FUNCTION_BLOCK FB_AnalogueInputBase IMPLEMENTS IAnalogueInput
VAR_INPUT
END_VAR
VAR_OUTPUT
END_VAR
VAR
	_processData : REFERENCE TO AnalogueStatus;
	_signalType : DINT;
	_resolution : DINT;
END_VAR

PROPERTY PUBLIC Error : bool
GET
Error := _processData.Underrange OR _processData.Overrange OR _processData.SyncError OR _processData.Error;
END_GET
END_PROPERTY

METHOD FB_init : BOOL
VAR_INPUT
	bInitRetains : BOOL; // if TRUE, the retain variables are initialized (warm start / cold start)
	bInCopyCode : BOOL;  // if TRUE, the instance afterwards gets moved into the copy code (online change)
	SignalType : SignalType;
	Resolution : Resolution;
	ProcessData : reference to AnalogueStatus;
END_VAR
CASE SignalType OF
	1: _signalType := 20;
	2: _signalType := 20;
	3: _signalType := 30;
	4: _signalType := 10;
END_CASE

CASE Resolution OF
	1: _resolution := 2048;
	2: _resolution := 32768;
	3: _resolution := 8388608;
END_CASE

_processData := ProcessData;
END_METHOD

METHOD GetConvertedValue : REAL
VAR
END_VAR
IF (_resolution = 0) OR (_signalType = 0) THEN
	RETURN;
END_IF

GetConvertedValue := _processData.Value * (_signalType/_resolution);
END_METHOD

METHOD GetRawValue : int
VAR_INPUT
END_VAR
GetRawValue := _processData.Value;
END_METHOD

END_FUNCTION_BLOCK

(* stored: Version 1.1.0.1, ProductVersion 3.1.4024.5
   POU FB_AnalogueInputBase: Id {ffe48a9a-1d37-40f8-b7a7-45cd91910e96}, SpecialFunc None
   Property Error: Id {79a5cfef-99b5-481c-81b7-13cb614e2233}
   Get Get: Id {51c26d9b-c891-4b59-82f1-015c97e0525e}
   Method FB_init: Id {e0500f8c-eb79-4e42-bb25-72de298c7e14}
   Method GetConvertedValue: Id {1d77c5be-2386-4642-9531-4f10dc497ecd}
   Method GetRawValue: Id {840f64bd-c848-40ab-944f-b870f219b250} *)
